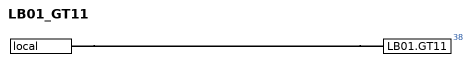
local := LB01.GT11;
ackFault S= local.ACK AND local.FAULT;
ackLal S= local.ACK AND local.LAL;
ackHal S= local.ACK AND local.HAL;
local.ACK R= true;
// Sensor error
AlarmAcknowledge01(
    Alarm := local.PV < -3200.0 AND NOT SYS_StartupDelayComm,
    InitPulse := SYS_InitPulse,
    AlarmAck := ackFault); // _BE_AlarmAckRemote
local.FAULT := AlarmAcknowledge01.AlarmActive;
// Deviation min/max
local.CSP1 := local.CSP - local.ADL;
local.CSP2 := local.CSP + local.ADL;
// Alarm Low
gt_Min(IN := local.PV < local.CSP1 AND NOT SYS_StartupDelayComm AND LB01.GeneralStart AND NOT local.FAULT, PT := DINT_TO_TIME(local.AD * 60000)); // TON
AlarmAcknowledge02(Alarm := gt_Min.Q, InitPulse := SYS_InitPulse, AlarmAck := ackLal); // _BE_AlarmAckRemote
local.LAL := AlarmAcknowledge02.AlarmActive;
// Alarm High
gt_Max(IN := local.PV > local.CSP2 AND NOT SYS_StartupDelayComm AND LB01.GeneralStart AND NOT local.FAULT, PT := DINT_TO_TIME(local.AD * 60000)); // TON
AlarmAcknowledge03(Alarm := gt_Max.Q, InitPulse := SYS_InitPulse, AlarmAck := ackHal); // _BE_AlarmAckRemote
local.HAL := AlarmAcknowledge03.AlarmActive;
// Status HMI
IF true THEN _w1 := 0; END_IF
local.Symbol := _w1;
_w2 := local.FAULT OR local.LAL OR local.HAL;
IF _w2 THEN _w3 := 2; END_IF
local.AL := _w2;
local.Symbol := _w3;
IF local.FAULT THEN _w4 := 3; END_IF
local.Symbol := _w4;
LB01.GT11 := local;
// al: input not connected

END_PROGRAM

// Device/AREA1/B001/LB01/Sensor/Temperature/GT21/LB01_GT21
PROGRAM LB01_GT21
VAR
	local:strSensor1;
	gt_Min: TON;
	gt_Max: TON;
	ackFault: BOOL;
	ackLal: BOOL;
	ackHal: BOOL;
	AlarmAcknowledge01: _BE_AlarmAckRemote;
	AlarmAcknowledge02: _BE_AlarmAckRemote;
	AlarmAcknowledge03: _BE_AlarmAckRemote;
END_VAR
VAR // added by the converter: edge detectors and wires of the graphical bodies
    _w1, _w3, _w4 : ANY;
    _w2 : BOOL;
END_VAR

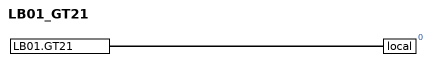
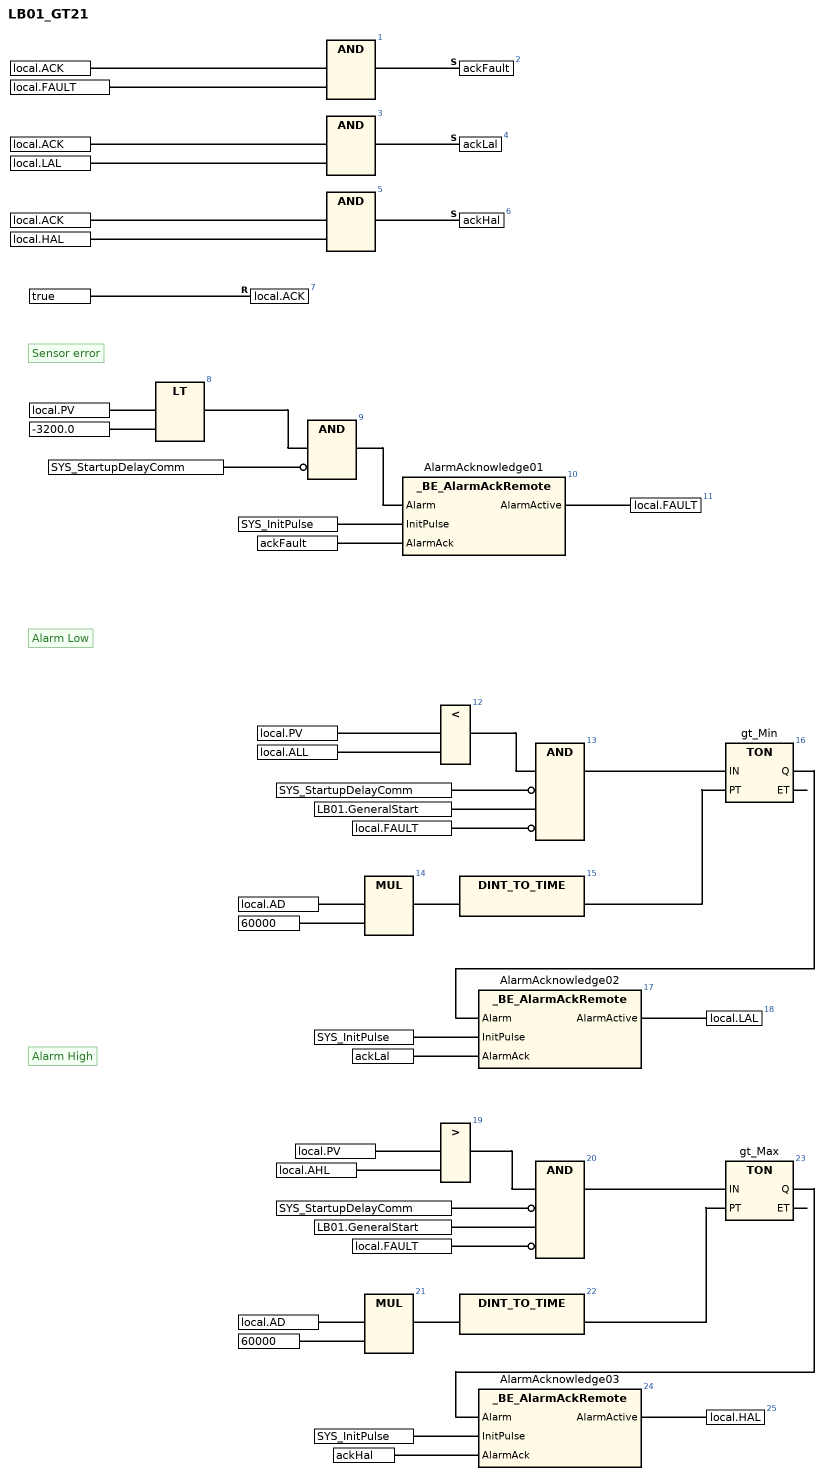
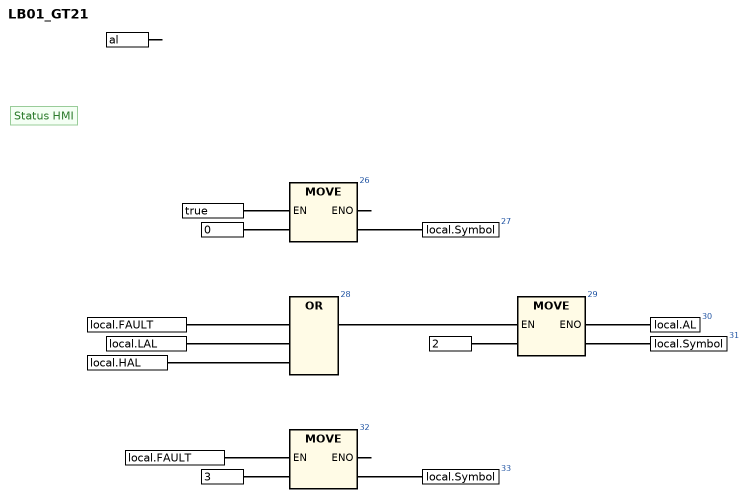
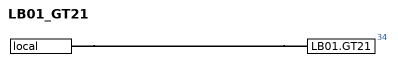
// note: 4 stored wires end on pins the file does not list and are not shown
local := LB01.GT21;
ackFault S= local.ACK AND local.FAULT;
ackLal S= local.ACK AND local.LAL;
ackHal S= local.ACK AND local.HAL;
local.ACK R= true;
// Sensor error
AlarmAcknowledge01(
    Alarm := local.PV < -3200.0 AND NOT SYS_StartupDelayComm,
    InitPulse := SYS_InitPulse,
    AlarmAck := ackFault); // _BE_AlarmAckRemote
local.FAULT := AlarmAcknowledge01.AlarmActive;
// Alarm Low
gt_Min(IN := local.PV < local.ALL AND NOT SYS_StartupDelayComm AND LB01.GeneralStart AND NOT local.FAULT, PT := DINT_TO_TIME(local.AD * 60000)); // TON
AlarmAcknowledge02(Alarm := gt_Min.Q, InitPulse := SYS_InitPulse, AlarmAck := ackLal); // _BE_AlarmAckRemote
local.LAL := AlarmAcknowledge02.AlarmActive;
// Alarm High
gt_Max(IN := local.PV > local.AHL AND NOT SYS_StartupDelayComm AND LB01.GeneralStart AND NOT local.FAULT, PT := DINT_TO_TIME(local.AD * 60000)); // TON
AlarmAcknowledge03(Alarm := gt_Max.Q, InitPulse := SYS_InitPulse, AlarmAck := ackHal); // _BE_AlarmAckRemote
local.HAL := AlarmAcknowledge03.AlarmActive;
// Status HMI
IF true THEN _w1 := 0; END_IF
local.Symbol := _w1;
_w2 := local.FAULT OR local.LAL OR local.HAL;
IF _w2 THEN _w3 := 2; END_IF
local.AL := _w2;
local.Symbol := _w3;
IF local.FAULT THEN _w4 := 3; END_IF
local.Symbol := _w4;
LB01.GT21 := local;
// al: input not connected

END_PROGRAM

// Device/AREA1/B001/LB01/Sensor/Temperature/GT41/LB01_GT41
PROGRAM LB01_GT41
VAR
	local:strSensor1;
	gt_Min: TON;
	gt_Max: TON;
	ackFault: BOOL;
	ackLal: BOOL;
	ackHal: BOOL;
	AlarmAcknowledg01: _BE_AlarmAckRemote;
	AlarmAcknowledge02: _BE_AlarmAckRemote;
	AlarmAcknowledge03: _BE_AlarmAckRemote;
END_VAR
VAR // added by the converter: edge detectors and wires of the graphical bodies
    _w1, _w3, _w4 : ANY;
    _w2 : BOOL;
END_VAR

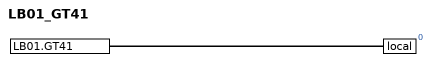
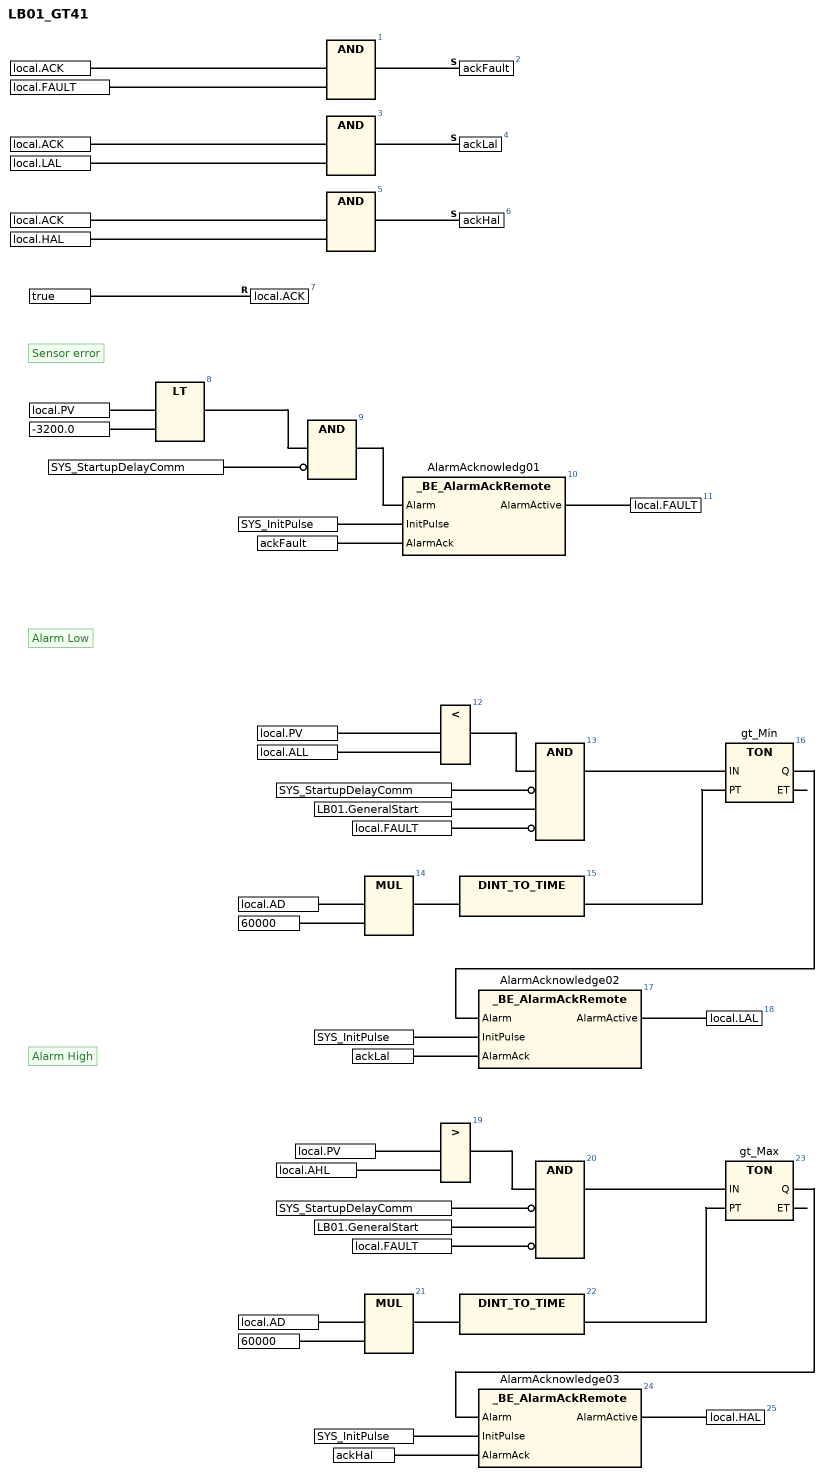
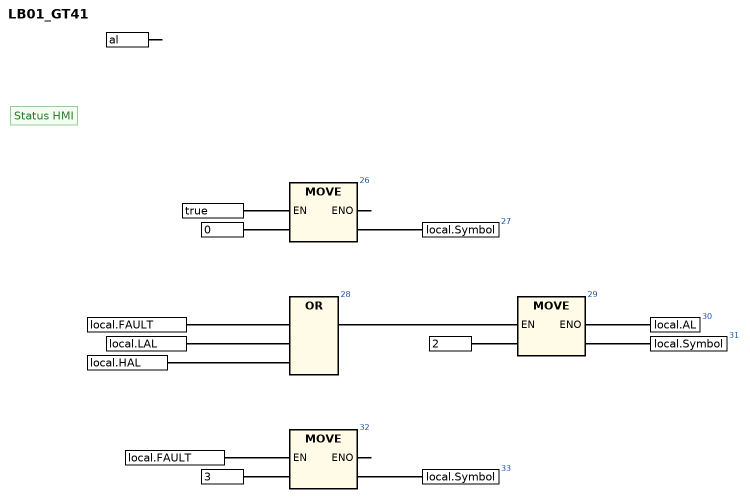
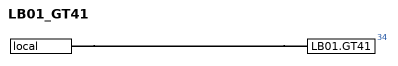
// note: 4 stored wires end on pins the file does not list and are not shown
local := LB01.GT41;
ackFault S= local.ACK AND local.FAULT;
ackLal S= local.ACK AND local.LAL;
ackHal S= local.ACK AND local.HAL;
local.ACK R= true;
// Sensor error
AlarmAcknowledg01(
    Alarm := local.PV < -3200.0 AND NOT SYS_StartupDelayComm,
    InitPulse := SYS_InitPulse,
    AlarmAck := ackFault); // _BE_AlarmAckRemote
local.FAULT := AlarmAcknowledg01.AlarmActive;
// Alarm Low
gt_Min(IN := local.PV < local.ALL AND NOT SYS_StartupDelayComm AND LB01.GeneralStart AND NOT local.FAULT, PT := DINT_TO_TIME(local.AD * 60000)); // TON
AlarmAcknowledge02(Alarm := gt_Min.Q, InitPulse := SYS_InitPulse, AlarmAck := ackLal); // _BE_AlarmAckRemote
local.LAL := AlarmAcknowledge02.AlarmActive;
// Alarm High
gt_Max(IN := local.PV > local.AHL AND NOT SYS_StartupDelayComm AND LB01.GeneralStart AND NOT local.FAULT, PT := DINT_TO_TIME(local.AD * 60000)); // TON
AlarmAcknowledge03(Alarm := gt_Max.Q, InitPulse := SYS_InitPulse, AlarmAck := ackHal); // _BE_AlarmAckRemote
local.HAL := AlarmAcknowledge03.AlarmActive;
// Status HMI
IF true THEN _w1 := 0; END_IF
local.Symbol := _w1;
_w2 := local.FAULT OR local.LAL OR local.HAL;
IF _w2 THEN _w3 := 2; END_IF
local.AL := _w2;
local.Symbol := _w3;
IF local.FAULT THEN _w4 := 3; END_IF
local.Symbol := _w4;
LB01.GT41 := local;
// al: input not connected

END_PROGRAM

// Device/AREA1/B001/LB01/Pump/P1/LB01_P1
PROGRAM LB01_P1
VAR
	local:strPumpExercise;
	fbControlPump2: _BE_Pump_2;
	fbPumpStartCondition: _BE_PumpStartConditions;
	fb_OperationalTime: _BE_OperationalTime;
	fbExercise: _BE_Exercise;
	ackAl01: BOOL;
	ackAl02: BOOL;
	sv_op: REAL;
	startPump: BOOL;
	AlarmFbAL01: _BE_AlarmAckRequired;
	AlarmFbAL02: _BE_AlarmAckRequired;
END_VAR
VAR // added by the converter: edge detectors and wires of the graphical bodies
    _w1 : ANY;
END_VAR

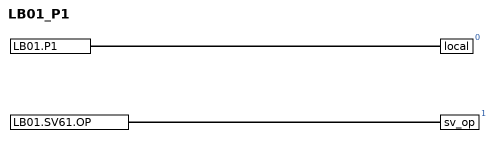
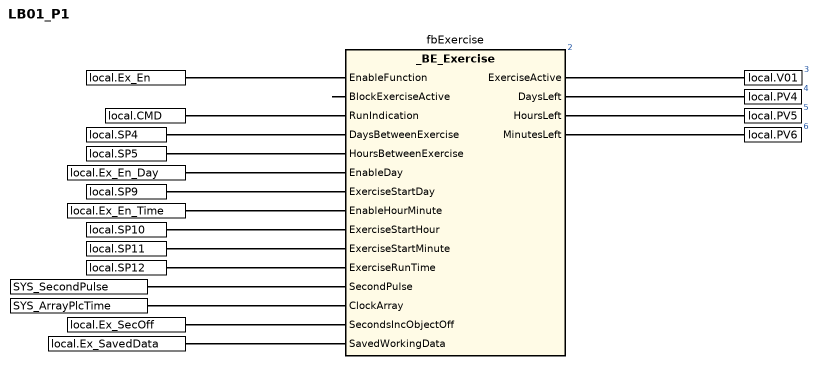
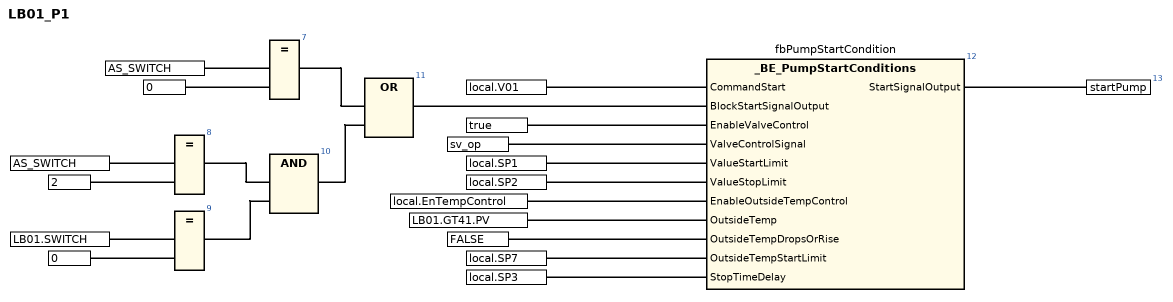
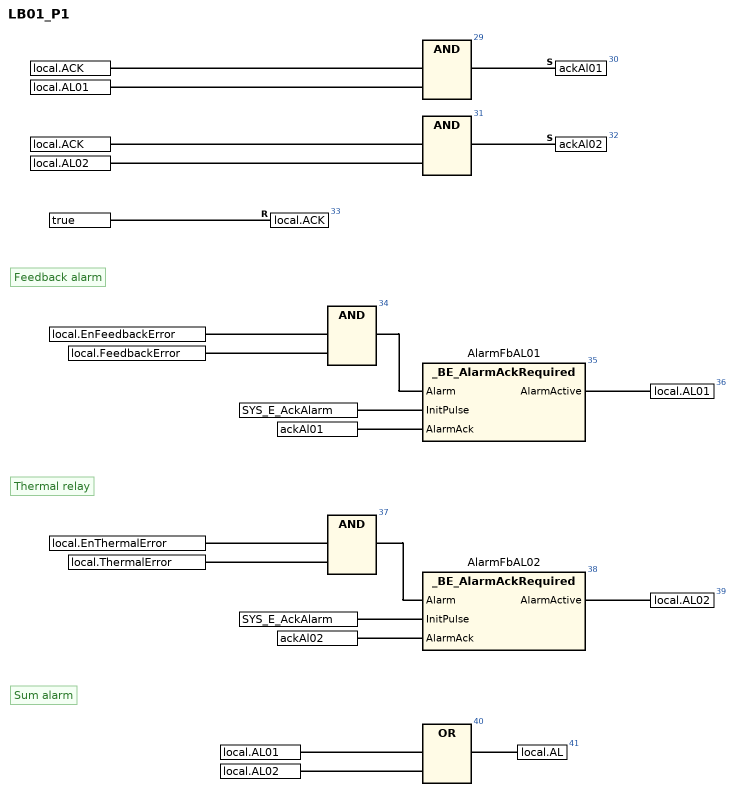
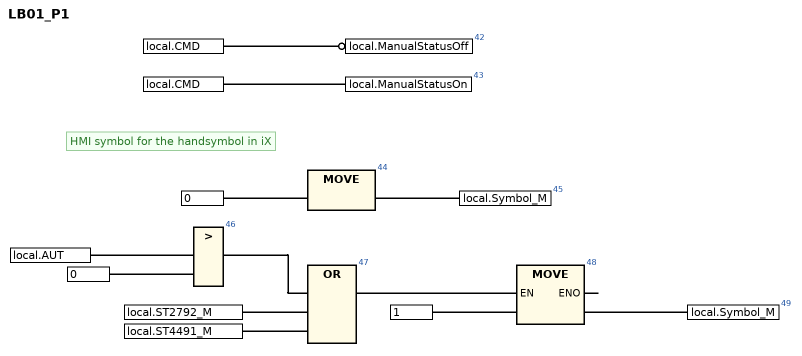
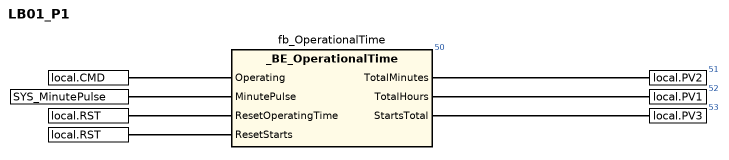
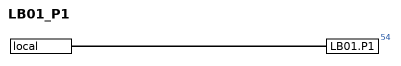
local := LB01.P1;
sv_op := LB01.SV61.OP;
fbExercise(
    EnableFunction := local.Ex_En,
    RunIndication := local.CMD,
    DaysBetweenExercise := local.SP4,
    HoursBetweenExercise := local.SP5,
    EnableDay := local.Ex_En_Day,
    ExerciseStartDay := local.SP9,
    EnableHourMinute := local.Ex_En_Time,
    ExerciseStartHour := local.SP10,
    ExerciseStartMinute := local.SP11,
    ExerciseRunTime := local.SP12,
    SecondPulse := SYS_SecondPulse,
    ClockArray := SYS_ArrayPlcTime,
    SecondsIncObjectOff := local.Ex_SecOff,
    SavedWorkingData := local.Ex_SavedData); // _BE_Exercise
local.V01 := fbExercise.ExerciseActive;
local.PV4 := fbExercise.DaysLeft;
local.PV5 := fbExercise.HoursLeft;
local.PV6 := fbExercise.MinutesLeft;
fbPumpStartCondition(
    CommandStart := local.V01,
    BlockStartSignalOutput := AS_SWITCH = 0 OR AS_SWITCH = 2 AND LB01.SWITCH = 0,
    EnableValveControl := true,
    ValveControlSignal := sv_op,
    ValueStartLimit := local.SP1,
    ValueStopLimit := local.SP2,
    EnableOutsideTempControl := local.EnTempControl,
    OutsideTemp := LB01.GT41.PV,
    OutsideTempDropsOrRise := FALSE,
    OutsideTempStartLimit := local.SP7,
    StopTimeDelay := local.SP3); // _BE_PumpStartConditions
startPump := fbPumpStartCondition.StartSignalOutput;
local.EnFeedbackError := local.SP6 > 0;
local.EnThermalError := local.SP8 > 0;
fbControlPump2(
    AutoStart := startPump,
    BlockAutoStart := false,
    RunIndication := local.V,
    EnableFeedbackAlarm := local.EnFeedbackError,
    FeedbackAlarmTimeDelay := local.SP6,
    EnableThermicRelayAlarm := local.EnThermalError,
    ThermicRelayOk := local.ThermicRelay,
    ThermicRelayAlarmTimeDelay := local.SP8,
    AlarmIndication := local.AL,
    AutoReg := local.AUT); // _BE_Pump_2
local.CMD := fbControlPump2.StartSignalOutput;
local.FeedbackError := fbControlPump2.FeedbackAlarm;
local.ThermalError := fbControlPump2.ThermicRelayAlarm;
// Manual control from hardware switches
local.Symbol := SEL(local.ST2792_M OR local.ST4491_M, fbControlPump2.Status, SEL(local.ST2792_MCMD OR local.ST4491_OPM > 0.5 AND local.ST4491_M, 0, 1));
ackAl01 S= local.ACK AND local.AL01;
ackAl02 S= local.ACK AND local.AL02;
local.ACK R= true;
// Feedback alarm
AlarmFbAL01(
    Alarm := local.EnFeedbackError AND local.FeedbackError,
    InitPulse := SYS_E_AckAlarm,
    AlarmAck := ackAl01); // _BE_AlarmAckRequired
local.AL01 := AlarmFbAL01.AlarmActive;
// Thermal relay
AlarmFbAL02(
    Alarm := local.EnThermalError AND local.ThermalError,
    InitPulse := SYS_E_AckAlarm,
    AlarmAck := ackAl02); // _BE_AlarmAckRequired
local.AL02 := AlarmFbAL02.AlarmActive;
// Sum alarm
local.AL := local.AL01 OR local.AL02;
local.ManualStatusOff := NOT local.CMD;
local.ManualStatusOn := local.CMD;
// HMI symbol for the handsymbol in iX
local.Symbol_M := 0;
IF local.AUT > 0 OR local.ST2792_M OR local.ST4491_M THEN _w1 := 1; END_IF
local.Symbol_M := _w1;
fb_OperationalTime(
    Operating := local.CMD,
    MinutePulse := SYS_MinutePulse,
    ResetOperatingTime := local.RST,
    ResetStarts := local.RST); // _BE_OperationalTime
local.PV2 := fb_OperationalTime.TotalMinutes;
local.PV1 := fb_OperationalTime.TotalHours;
local.PV3 := fb_OperationalTime.StartsTotal;
LB01.P1 := local;

END_PROGRAM

// Device/AREA1/B001/LB01/Fan/TF1/LB01_TF1_Analog
PROGRAM LB01_TF1_Analog
VAR
	local:strFan_Analog;
	localGP:strSensor2_Regulator;
	ControlFan: _BE_Fan;
	FbRegulator: _BE_Regulator;
	_BE_Fan2: _BE_Fan_2;
	reset_en: RS;
	AlarmFbAl01: _BE_AlarmAckRequired;
	AlarmFbAl02: _BE_AlarmAckRequired;
	fb_OperationalTime: _BE_OperationalTime;
	ackAl01: BOOL;
	ackAl02: BOOL;
	fanGuardOk: BOOL;
END_VAR
VAR // added by the converter: edge detectors and wires of the graphical bodies
    _w1, _w3, _w4, _w5 : ANY;
    _w2 : BOOL;
END_VAR

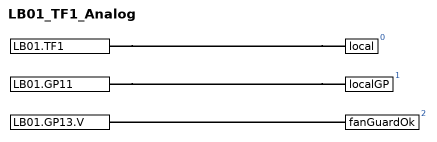
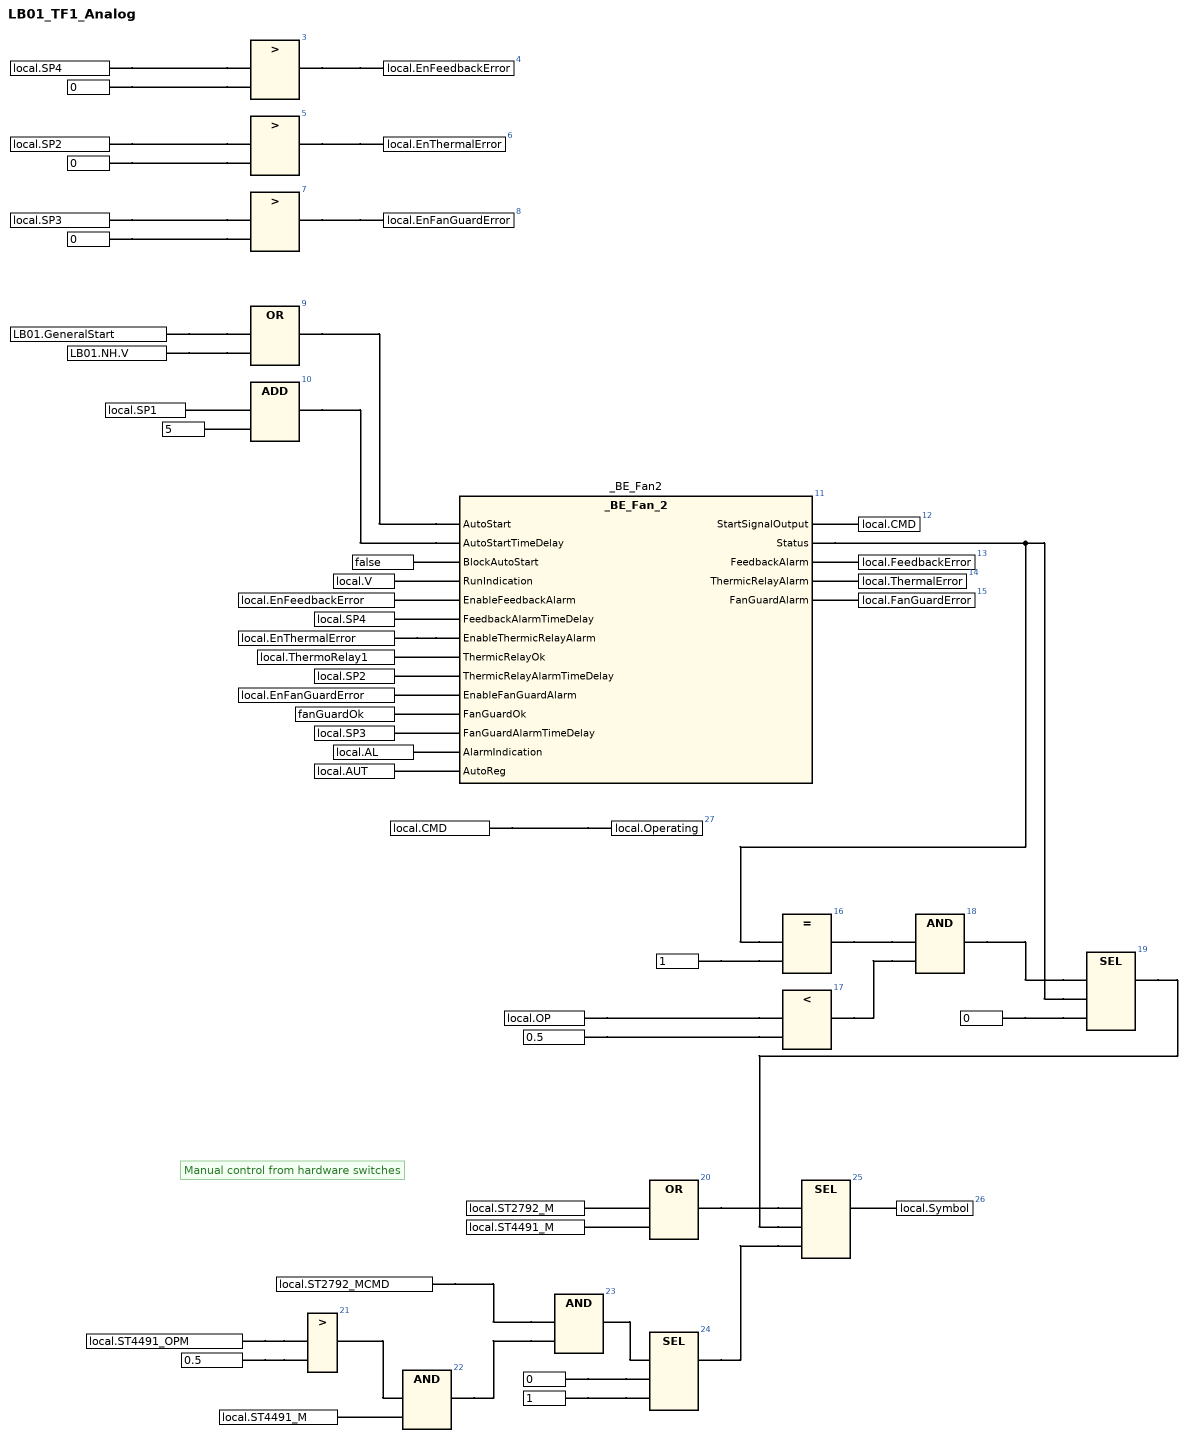
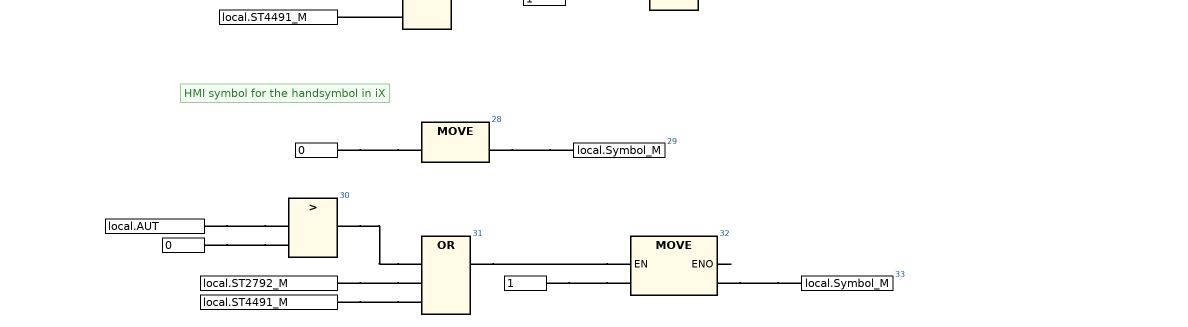
